{attribute addProperty BoxType "EP2316-0008-0018"}
{attribute addProperty Id "DIG_InputsAT %I*DIG_Inputs_9F71B9E27290DIG_Diag_InputsAT %I*DIG_Diag_Inputs_AC4A9AF06480DIG_Inputs_DeviceAT %I*DIG_Inputs_Device_213DCE554050DIG_OutputsAT %Q*DIG_Outputs_33B763766480DIG_Outputs_DeviceAT %Q*DIG_Outputs_Device_735003021620WcStateAT %I*WcState_F855686C1620InfoDataAT %I*InfoData_BC63D37F80100"}
{attribute addProperty CRC "2060676949"}
{attribute addProperty SizeInBites "352"}
{attribute addProperty SizeInBytes "44"}
TYPE EP2316_51C6E99B :
STRUCT
	{attribute addProperty Name "DIG_Inputs"}
	DIG_Inputs : DIG_Inputs_9F71B9E2;
	{attribute addProperty Name "DIG_Diag_Inputs"}
	DIG_Diag_Inputs : DIG_Diag_Inputs_AC4A9AF0;
	{attribute addProperty Name "DIG_Inputs_Device"}
	DIG_Inputs_Device : DIG_Inputs_Device_213DCE55;
	{attribute addProperty Name "DIG_Outputs"}
	DIG_Outputs : DIG_Outputs_33B76376;
	{attribute addProperty Name "DIG_Outputs_Device"}
	DIG_Outputs_Device : DIG_Outputs_Device_73500302;
	{attribute addProperty Name "WcState"}
	WcState : WcState_F855686C;
	{attribute addProperty Name "InfoData"}
	InfoData : InfoData_BC63D37F;
END_STRUCT
END_TYPE

(* stored: Version 1.2.0.0, ProductVersion 3.1.4024.9
   DUT EP2316_51C6E99B: Id {0309aef1-289c-412c-b6d3-5ba79ed79f2e} *)
